Universal Robots PolyScope program: c_to_d.urp

Program c_to_d (installation=string_planes directory=/programs/string_crossings createdIn=5.17.3 lastSavedIn=5.17.3 robotSerialNumber=20245501435)
Calibrated DH parameters: a=[0.000154, -0.137004, -0.385524, -0.00002, 0.000092, 0]; d=[0.162441, 211.794786, -230.585024, 18.923638, 0.099786, 0.09951]; alpha=[1.569493, -0.001902, 0.003874, 1.570111, -1.570167, 0]; deltaTheta=[0, -1.242934, 1.056292, 0.186646, 0.000002, 0.000001]
InitVariablesNode
Robot Program (runOnlyOnce=false)
  bow_section := -1
  If bow_section≟-1
    MoveJ speed 60 deg/s, acceleration 80 deg/s^2 (useActiveTCP=true) feature=Base
      Waypoint Waypoint_2 (Relative): relativeFromPosition TCP in base x=245.287 y=570.708 z=53.279 mm, rx=-1.8425 ry=-1.3918 rz=0.0687 rad; joints [-132.226, -24.799, 96.314, -169.323, -42.69, -112.608] deg; TCP offset x=28.21 y=-96.107 z=-99.69 mm, rx=0 ry=0 rz=0 rad; TCP in base x=316.071 y=723.616 z=117.783 mm, rx=-1.5349 ry=-2.2386 rz=1.1275 rad; joints [-128.458, -21.868, 50.821, -72.931, -81.953, -152.853] deg
  ElseIf bow_section≟0
    MoveJ speed 60 deg/s, acceleration 80 deg/s^2 (useActiveTCP=true) feature=Base
      Waypoint Waypoint_1 (Relative): relativeFromPosition TCP in base x=195.299 y=411.479 z=21.277 mm, rx=-1.7342 ry=-1.517 rz=0.432 rad; joints [-140.233, -30.937, 122.528, -154.99, -45.802, -143.198] deg; TCP in base x=337.286 y=452.569 z=146.265 mm, rx=-1.6084 ry=-2.1978 rz=1.0429 rad; joints [-146.229, -47.168, 100.749, -99.804, -91.441, -163.024] deg
  Else 
    MoveJ speed 60 deg/s, acceleration 80 deg/s^2 (useActiveTCP=true) feature=Base
      Waypoint Waypoint_3 (Relative): relativeFromPosition TCP in base x=152.636 y=275.828 z=-5.99 mm, rx=-1.6121 ry=-1.6008 rz=0.7404 rad; joints [-153.501, -26.652, 138.519, -151.349, -62.643, -165.795] deg; TCP in base x=340.805 y=238.622 z=127.329 mm, rx=-1.5375 ry=-2.1223 rz=1.0863 rad; joints [-167.854, -53.467, 123.568, -113.681, -104.544, -179.467] deg
